// Mitsubishi GX Works2 project: timer+sequence_2   PLC: Q03UDV

PROGRAM MAIN
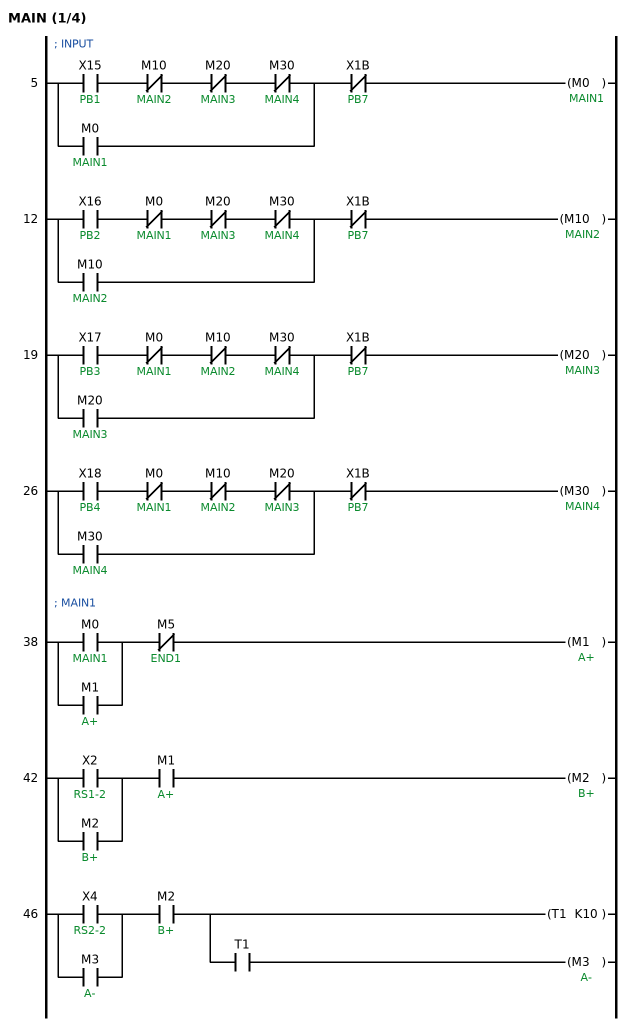
; INPUT
5     LD      X15  ; PB1
      ANI     M10  ; MAIN2
      ANI     M20  ; MAIN3
      ANI     M30  ; MAIN4
      OR      M0  ; MAIN1
      ANI     X1B  ; PB7
      OUT     M0  ; MAIN1
12    LD      X16  ; PB2
      ANI     M0  ; MAIN1
      ANI     M20  ; MAIN3
      ANI     M30  ; MAIN4
      OR      M10  ; MAIN2
      ANI     X1B  ; PB7
      OUT     M10  ; MAIN2
19    LD      X17  ; PB3
      ANI     M0  ; MAIN1
      ANI     M10  ; MAIN2
      ANI     M30  ; MAIN4
      OR      M20  ; MAIN3
      ANI     X1B  ; PB7
      OUT     M20  ; MAIN3
26    LD      X18  ; PB4
      ANI     M0  ; MAIN1
      ANI     M10  ; MAIN2
      ANI     M20  ; MAIN3
      OR      M30  ; MAIN4
      ANI     X1B  ; PB7
      OUT     M30  ; MAIN4
; MAIN1
38    LD      M0  ; MAIN1
      OR      M1  ; A+
      ANI     M5  ; END1
      OUT     M1  ; A+
42    LD      X2  ; RS1-2
      OR      M2  ; B+
      AND     M1  ; A+
      OUT     M2  ; B+
46    LD      X4  ; RS2-2
      OR      M3  ; A-
      AND     M2  ; B+
      OUT     T1 K10
      AND     T1
      OUT     M3  ; A-
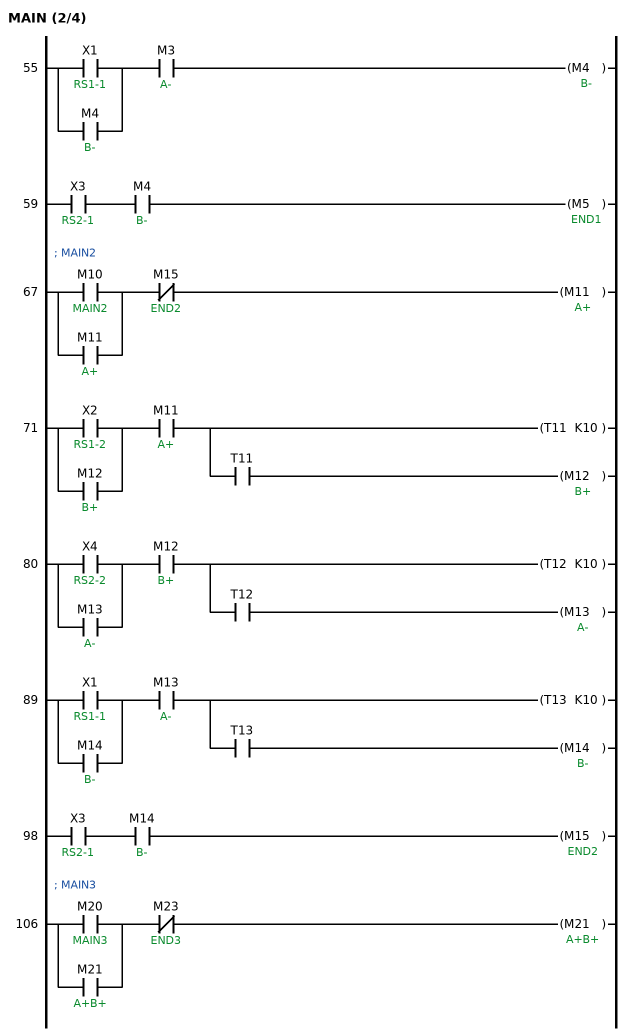
55    LD      X1  ; RS1-1
      OR      M4  ; B-
      AND     M3  ; A-
      OUT     M4  ; B-
59    LD      X3  ; RS2-1
      AND     M4  ; B-
      OUT     M5  ; END1
; MAIN2
67    LD      M10  ; MAIN2
      OR      M11  ; A+
      ANI     M15  ; END2
      OUT     M11  ; A+
71    LD      X2  ; RS1-2
      OR      M12  ; B+
      AND     M11  ; A+
      OUT     T11 K10
      AND     T11
      OUT     M12  ; B+
80    LD      X4  ; RS2-2
      OR      M13  ; A-
      AND     M12  ; B+
      OUT     T12 K10
      AND     T12
      OUT     M13  ; A-
89    LD      X1  ; RS1-1
      OR      M14  ; B-
      AND     M13  ; A-
      OUT     T13 K10
      AND     T13
      OUT     M14  ; B-
98    LD      X3  ; RS2-1
      AND     M14  ; B-
      OUT     M15  ; END2
; MAIN3
106   LD      M20  ; MAIN3
      OR      M21  ; A+B+
      ANI     M23  ; END3
      OUT     M21  ; A+B+
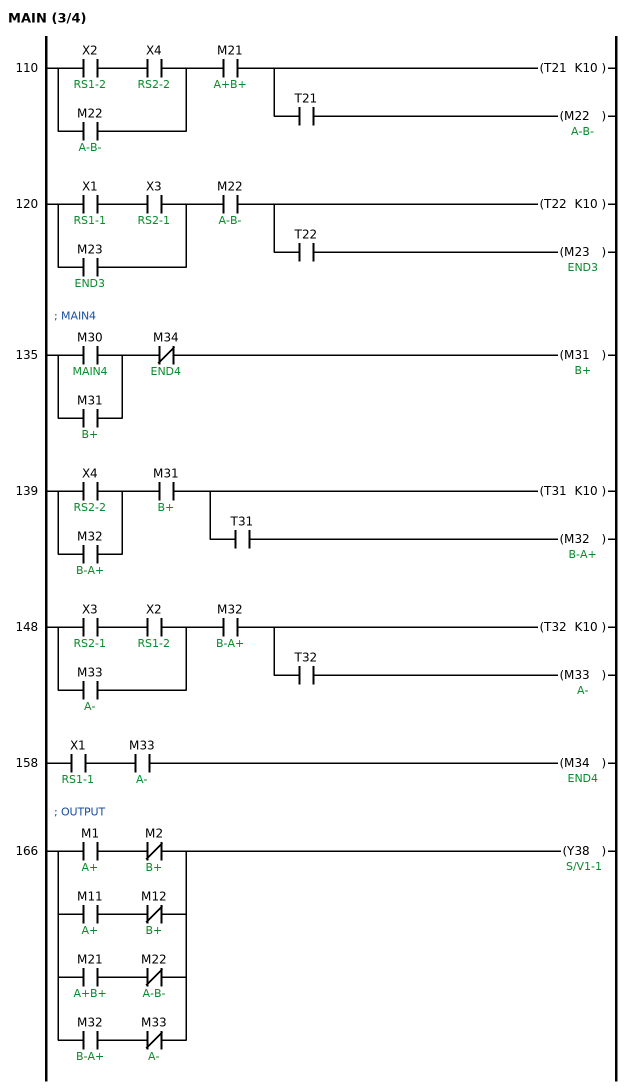
110   LD      X2  ; RS1-2
      AND     X4  ; RS2-2
      OR      M22  ; A-B-
      AND     M21  ; A+B+
      OUT     T21 K10
      AND     T21
      OUT     M22  ; A-B-
120   LD      X1  ; RS1-1
      AND     X3  ; RS2-1
      OR      M23  ; END3
      AND     M22  ; A-B-
      OUT     T22 K10
      AND     T22
      OUT     M23  ; END3
; MAIN4
135   LD      M30  ; MAIN4
      OR      M31  ; B+
      ANI     M34  ; END4
      OUT     M31  ; B+
139   LD      X4  ; RS2-2
      OR      M32  ; B-A+
      AND     M31  ; B+
      OUT     T31 K10
      AND     T31
      OUT     M32  ; B-A+
148   LD      X3  ; RS2-1
      AND     X2  ; RS1-2
      OR      M33  ; A-
      AND     M32  ; B-A+
      OUT     T32 K10
      AND     T32
      OUT     M33  ; A-
158   LD      X1  ; RS1-1
      AND     M33  ; A-
      OUT     M34  ; END4
; OUTPUT
166   LD      M1  ; A+
      ANI     M2  ; B+
      LD      M11  ; A+
      ANI     M12  ; B+
      ORB
      LD      M21  ; A+B+
      ANI     M22  ; A-B-
      ORB
      LD      M32  ; B-A+
      ANI     M33  ; A-
      ORB
      OUT     Y38  ; S/V1-1
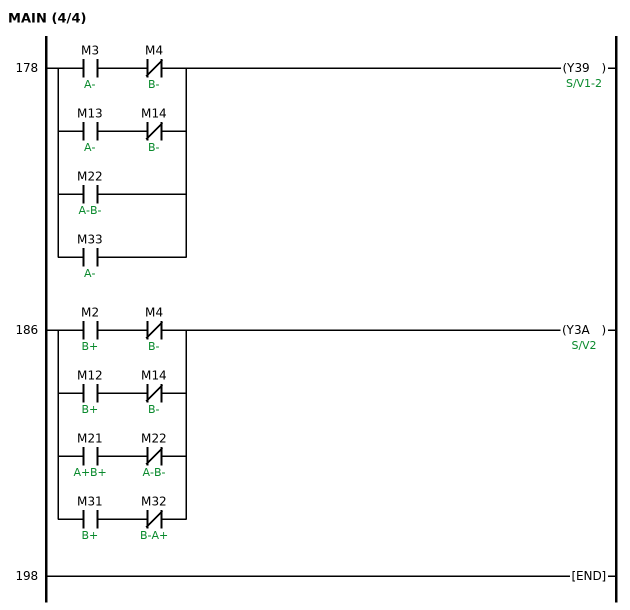
178   LD      M3  ; A-
      ANI     M4  ; B-
      LD      M13  ; A-
      ANI     M14  ; B-
      ORB
      OR      M22  ; A-B-
      OR      M33  ; A-
      OUT     Y39  ; S/V1-2
186   LD      M2  ; B+
      ANI     M4  ; B-
      LD      M12  ; B+
      ANI     M14  ; B-
      ORB
      LD      M21  ; A+B+
      ANI     M22  ; A-B-
      ORB
      LD      M31  ; B+
      ANI     M32  ; B-A+
      ORB
      OUT     Y3A  ; S/V2
198   END
END_PROGRAM
